PROGRAM UDPTest
VAR
	socketCreate:	FB_SocketUdpCreate;
	socketSend:		FB_SocketUdpSendTo;
	createNow: 		BOOL;
	sendNow:		BOOL;
	sMsg:			STRING[20] := 'Hello World';
	configCreate: 	BOOL := true;
END_VAR




IF configCreate THEN
	socketCreate.sSrvNetId := '39.19.23.23.1.1';
	socketCreate.sLocalHost := '192.168.56.101';
	socketCreate.nLocalPort := 41414;
	socketCreate.tTimeout := T#5S;
	configCreate := FALSE;
END_IF


//IF createNow THEN
	socketCreate.bExecute := createNow;
//	createNow := FALSE;
//END_IF


socketSend.hSocket := socketCreate.hSocket;
socketSend.sSrvNetId := '';
socketSend.sRemoteHost := '192.168.56.1';
socketSend.nRemotePort := 8000;
socketSend.cbLen := LEN(sMsg);
socketSend.pSrc := ADR(sMsg);
socketSend.tTimeout := T#5S;

IF sendNow THEN
	socketSend.bExecute := sendNow;
	sendNow := FALSE;
END_IF

// CAll fbs
socketCreate();
socketSend();

END_PROGRAM

(* stored: Version 1.1.0.1, ProductVersion 3.1.4024.12
   POU UDPTest: Id {d4ea590e-d88c-4479-a1c6-26e991dfdda3}, SpecialFunc None *)
